// TIA Portal V18 export
TYPE "typeMotPara"
// stored: IsFailsafeCompliant false
   STRUCT
      t_acc_50Hz_USER : Real;
      v_absoluteMax_LOGIC : Real;
      dist_absMax_LOGIC : Real;
      v_crawl_USER : Real;
      dist_crawl_USER : Real;
      dist_stop_USER : Real;
      dist_auto_done_LOGIC : Real;
      pos_calib_USER : Real;
      pos_lim_fwd_USER : Real;
      pos_lim_rev_USER : Real;
      v_blind_USER : Real;
      v_manual_USER : Real;
      v_auto_USER : Real;
      t_er : Time := T#3s;
   END_STRUCT;
END_TYPE
